{attribute 'enable_dynamic_creation'}
FUNCTION_BLOCK FB_Triangle IMPLEMENTS I_Shape
VAR_INPUT
END_VAR
VAR_OUTPUT
END_VAR
VAR
END_VAR

{warning 'Agregar implementación de método'}
METHOD M_Draw : BOOL
ADSLOGSTR(ADSLOG_MSGTYPE_HINT, 'Draw Triangle', '');
M_Draw := TRUE;
END_METHOD

END_FUNCTION_BLOCK

(* stored: Version 1.1.0.1, ProductVersion 3.1.4024.12
   POU FB_Triangle: Id {2edf1aa3-0e4d-4a4e-8b70-2fd8e2fb2a4f}, SpecialFunc None
   Method M_Draw: Id {0e549d57-17d0-4a5b-b18f-4fb7f8cc88de} *)
